{attribute wpf [Container(Layout.Tabs)]}
TYPE LayoutTabsStruct EXTENDS VariousTypesStruct :
STRUCT
END_STRUCT
END_TYPE

(* stored: Version 1.1.0.1, ProductVersion 3.1.4024.9
   DUT LayoutTabsStruct: Id {6c17bf70-7c0a-4257-8c27-ce0eac3180c5} *)
